# EPICS substitutions: FINS/FINS-IOC-01App/Db/imat-plc-attn.substitutions
file "$(TOP)/FINS-IOC-01App/Db/imat-plc-header.template" {
	{ P=\$(P), Q=\$(Q) }
}

file "$(TOP)/FINS-IOC-01App/Db/imat-plc-attn-main.template" {
	{ P=\$(P), Q=\$(Q) }
}
